RESOURCE RES0 : EMB_RES_ECO
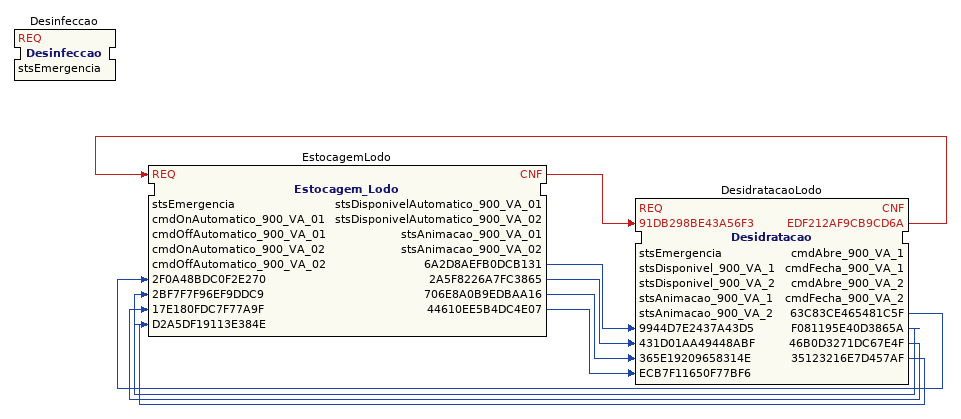
  FBS
    EstocagemLodo : Estocagem_Lodo;
    DesidratacaoLodo : Desidratacao;
    Desinfeccao : Desinfeccao;
  END_FBS
  EVENT_CONNECTIONS
    EstocagemLodo.CNF TO DesidratacaoLodo.91DB298BE43A56F3;
    DesidratacaoLodo.EDF212AF9CB9CD6A TO EstocagemLodo.REQ;
  END_CONNECTIONS
  DATA_CONNECTIONS
    EstocagemLodo.6A2D8AEFB0DCB131 TO DesidratacaoLodo.9944D7E2437A43D5;
    EstocagemLodo.2A5F8226A7FC3865 TO DesidratacaoLodo.431D01AA49448ABF;
    EstocagemLodo.706E8A0B9EDBAA16 TO DesidratacaoLodo.365E19209658314E;
    EstocagemLodo.44610EE5B4DC4E07 TO DesidratacaoLodo.ECB7F11650F77BF6;
    DesidratacaoLodo.63C83CE465481C5F TO EstocagemLodo.2F0A48BDC0F2E270;
    DesidratacaoLodo.F081195E40D3865A TO EstocagemLodo.2BF7F7F96EF9DDC9;
    DesidratacaoLodo.46B0D3271DC67E4F TO EstocagemLodo.17E180FDC7F77A9F;
    DesidratacaoLodo.35123216E7D457AF TO EstocagemLodo.D2A5DF19113E384E;
  END_CONNECTIONS
END_RESOURCE
